{attribute 'qualified_only'}
VAR_GLOBAL
	VTD_Sys:  ARRAY[1..2] OF VTD_Settings_DUT;
	ECnv_Sys:  ARRAY[1..2] OF ECnv_Settings_DUT;
	LCnv_Sys:  ARRAY[1..2] OF Cnv_VTD_Settings_DUT;
// 	Shuttle_MQTT:  MQTT_Settings;
	System:  System_Settings_DUT;
END_VAR

(* stored: Version 1.1.0.1
   GVL Settings: Id {9b82498a-e9a0-4bb6-a6fe-ce7c787e0820} *)
